INTERFACE I_SessionIdGenerator

METHOD PUBLIC Generate : T_MAXSTRING
VAR_INPUT
END_VAR
END_METHOD

END_INTERFACE

(* stored: Version 1.1.0.1, ProductVersion 3.1.4024.12
   Itf I_SessionIdGenerator: Id {ad7f292d-bd17-06c4-00f1-6e77a025a762}
   Method Generate: Id {b5bb1dfd-ab5d-0b34-0d79-b9b26e879888} *)
